Fanuc TP program (LS listing): DISTI_LINE_V10.LS

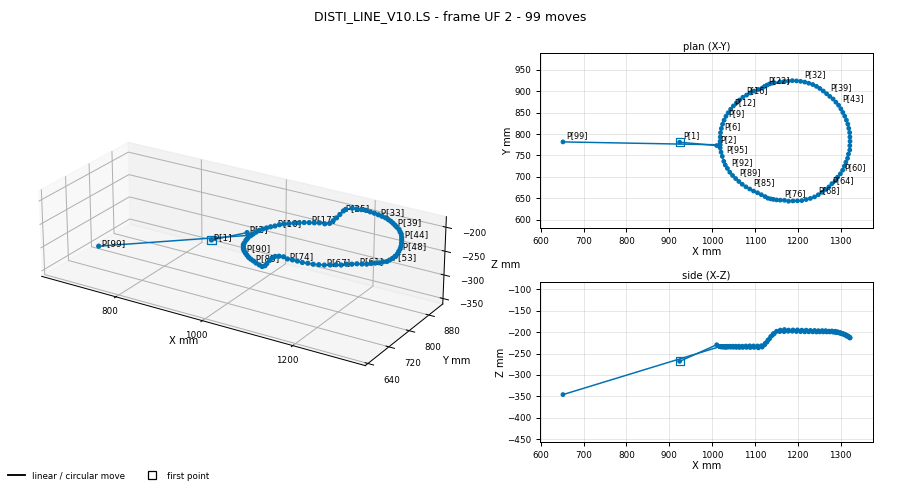
[picture p0: tool path of DISTI_LINE_V10.LS in frame UF 2, 99 of 99 moves have a stored position in this frame; points joined in program order, loops and branches not executed]
/PROG  DISTI_LINE_V10
/ATTR
OWNER		= MNEDITOR;
COMMENT		= "WeldPRO Auto-Gen";
PROG_SIZE	= 7125;
CREATE		= DATE 26-07-31  TIME 11:19:16;
MODIFIED	= DATE 26-07-31  TIME 13:58:52;
FILE_NAME	= DISTI_LI;
VERSION		= 0;
LINE_COUNT	= 113;
MEMORY_SIZE	= 7445;
PROTECT		= READ_WRITE;
TCD:  STACK_SIZE	= 0,
      TASK_PRIORITY	= 50,
      TIME_SLICE	= 0,
      BUSY_LAMP_OFF	= 0,
      ABORT_REQUEST	= 0,
      PAUSE_REQUEST	= 0;
DEFAULT_GROUP	= 1,*,*,*,*;
CONTROL_CODE	= 00000000 00000000;
/APPL
/MN
   1:  !WeldPRO Auto-Generated TPP ;
   2:  !TOR_XL_2026, TOR_xl_2907 ;
   3:   ;
   4:  UFRAME_NUM=2 ;
   5:  UTOOL_NUM=2 ;
   6:  !Feature Approach ;
   7:J P[1] 100% FINE    ;
   8:   ;
   9:  !Segment1 ;
  10:L P[2] 2000mm/sec FINE    ;
  11:   ;
  12:  CALL LASER_OFF    ;
  13:L P[3] R[23:moving]mm/sec CNT100    ;
  14:L P[4] R[23:moving]mm/sec CNT100    ;
  15:L P[5] R[23:moving]mm/sec CNT100    ;
  16:L P[6] R[23:moving]mm/sec CNT100    ;
  17:L P[7] R[23:moving]mm/sec CNT100    ;
  18:L P[8] R[23:moving]mm/sec CNT100    ;
  19:L P[9] R[23:moving]mm/sec CNT100    ;
  20:L P[10] R[23:moving]mm/sec CNT100    ;
  21:L P[11] R[23:moving]mm/sec CNT100    ;
  22:L P[12] R[23:moving]mm/sec CNT100    ;
  23:L P[13] R[23:moving]mm/sec CNT100    ;
  24:L P[14] R[23:moving]mm/sec CNT100    ;
  25:L P[15] R[23:moving]mm/sec CNT100    ;
  26:L P[16] R[23:moving]mm/sec CNT100    ;
  27:L P[17] R[23:moving]mm/sec CNT100    ;
  28:L P[18] R[23:moving]mm/sec CNT100    ;
  29:L P[19] R[23:moving]mm/sec CNT100    ;
  30:L P[20] R[23:moving]mm/sec CNT100    ;
  31:L P[21] R[23:moving]mm/sec CNT100    ;
  32:L P[22] R[23:moving]mm/sec CNT100    ;
  33:L P[23] R[23:moving]mm/sec CNT100    ;
  34:L P[24] R[23:moving]mm/sec CNT100    ;
  35:L P[25] R[23:moving]mm/sec CNT100    ;
  36:L P[26] R[23:moving]mm/sec CNT100    ;
  37:L P[27] R[23:moving]mm/sec CNT100    ;
  38:L P[28] R[23:moving]mm/sec CNT100    ;
  39:L P[29] R[23:moving]mm/sec CNT100    ;
  40:L P[30] R[23:moving]mm/sec CNT100    ;
  41:L P[31] R[23:moving]mm/sec CNT100    ;
  42:L P[32] R[23:moving]mm/sec CNT100    ;
  43:L P[33] R[23:moving]mm/sec CNT100    ;
  44:L P[34] R[23:moving]mm/sec CNT100    ;
  45:L P[35] R[23:moving]mm/sec CNT100    ;
  46:L P[36] R[23:moving]mm/sec CNT100    ;
  47:L P[37] R[23:moving]mm/sec CNT100    ;
  48:L P[38] R[23:moving]mm/sec CNT100    ;
  49:L P[39] R[23:moving]mm/sec CNT100    ;
  50:L P[40] R[23:moving]mm/sec CNT100    ;
  51:L P[41] R[23:moving]mm/sec CNT100    ;
  52:L P[42] R[23:moving]mm/sec CNT100    ;
  53:L P[43] R[23:moving]mm/sec CNT100    ;
  54:L P[44] R[23:moving]mm/sec CNT100    ;
  55:L P[45] R[23:moving]mm/sec CNT100    ;
  56:L P[46] R[23:moving]mm/sec CNT100    ;
  57:L P[47] R[23:moving]mm/sec CNT100    ;
  58:L P[48] R[23:moving]mm/sec CNT100    ;
  59:L P[49] R[23:moving]mm/sec CNT100    ;
  60:L P[50] R[23:moving]mm/sec CNT100    ;
  61:L P[51] R[23:moving]mm/sec CNT100    ;
  62:L P[52] R[23:moving]mm/sec CNT100    ;
  63:L P[53] R[23:moving]mm/sec CNT100    ;
  64:L P[54] R[23:moving]mm/sec CNT100    ;
  65:L P[55] R[23:moving]mm/sec CNT100    ;
  66:L P[56] R[23:moving]mm/sec CNT100    ;
  67:L P[57] R[23:moving]mm/sec CNT100    ;
  68:L P[58] R[23:moving]mm/sec CNT100    ;
  69:L P[59] R[23:moving]mm/sec CNT100    ;
  70:L P[60] R[23:moving]mm/sec CNT100    ;
  71:L P[61] R[23:moving]mm/sec CNT100    ;
  72:L P[62] R[23:moving]mm/sec CNT100    ;
  73:L P[63] R[23:moving]mm/sec CNT100    ;
  74:L P[64] R[23:moving]mm/sec CNT100    ;
  75:L P[65] R[23:moving]mm/sec CNT100    ;
  76:L P[66] R[23:moving]mm/sec CNT100    ;
  77:L P[67] R[23:moving]mm/sec CNT100    ;
  78:L P[68] R[23:moving]mm/sec CNT100    ;
  79:L P[69] R[23:moving]mm/sec CNT100    ;
  80:L P[70] R[23:moving]mm/sec CNT100    ;
  81:L P[71] R[23:moving]mm/sec CNT100    ;
  82:L P[72] R[23:moving]mm/sec CNT100    ;
  83:L P[73] R[23:moving]mm/sec CNT100    ;
  84:L P[74] R[23:moving]mm/sec CNT100    ;
  85:L P[75] R[23:moving]mm/sec CNT100    ;
  86:L P[76] R[23:moving]mm/sec CNT100    ;
  87:L P[77] R[23:moving]mm/sec CNT100    ;
  88:L P[78] R[23:moving]mm/sec CNT100    ;
  89:L P[79] R[23:moving]mm/sec CNT100    ;
  90:L P[80] R[23:moving]mm/sec CNT100    ;
  91:L P[81] R[23:moving]mm/sec CNT100    ;
  92:L P[82] R[23:moving]mm/sec CNT100    ;
  93:L P[83] R[23:moving]mm/sec CNT100    ;
  94:L P[84] R[23:moving]mm/sec CNT100    ;
  95:L P[85] R[23:moving]mm/sec CNT100    ;
  96:L P[86] R[23:moving]mm/sec CNT100    ;
  97:L P[87] R[23:moving]mm/sec CNT100    ;
  98:L P[88] R[23:moving]mm/sec CNT100    ;
  99:L P[89] R[23:moving]mm/sec CNT100    ;
 100:L P[90] R[23:moving]mm/sec CNT100    ;
 101:L P[91] R[23:moving]mm/sec CNT100    ;
 102:L P[92] R[23:moving]mm/sec CNT100    ;
 103:L P[93] R[23:moving]mm/sec CNT100    ;
 104:L P[94] R[23:moving]mm/sec CNT100    ;
 105:L P[95] R[23:moving]mm/sec CNT100    ;
 106:L P[96] R[23:moving]mm/sec CNT100    ;
 107:L P[97] R[23:moving]mm/sec CNT100    ;
 108:L P[98] R[23:moving]mm/sec FINE    ;
 109:  CALL LASER_OFF    ;
 110:   ;
 111:  !Feature Retreat ;
 112:L P[99] 2000mm/sec FINE    ;
 113:  CALL ROTATE    ;
/POS
P[1]{
   GP1:
	UF : 2, UT : 2,		CONFIG : 'F D T, 0, 0, 0',
	X =   924.335  mm,	Y =   780.986  mm,	Z =  -268.284  mm,
	W =  -106.495 deg,	P =   -15.000 deg,	R =    94.234 deg
};
P[2]{
   GP1:
	UF : 2, UT : 2,		CONFIG : 'F D T, 0, 0, 0',
	X =  1011.104  mm,	Y =   773.115  mm,	Z =  -229.520  mm,
	W =  -106.497 deg,	P =   -14.995 deg,	R =    94.216 deg
};
P[3]{
   GP1:
	UF : 2, UT : 2,		CONFIG : 'F D T, 0, 0, 0',
	X =  1018.942  mm,	Y =   775.004  mm,	Z =  -233.963  mm,
	W =  -106.501 deg,	P =   -14.998 deg,	R =    94.232 deg
};
P[4]{
   GP1:
	UF : 2, UT : 2,		CONFIG : 'F D T, 0, 0, 0',
	X =  1018.850  mm,	Y =   783.088  mm,	Z =  -234.009  mm,
	W =  -106.497 deg,	P =   -15.098 deg,	R =    90.375 deg
};
P[5]{
   GP1:
	UF : 2, UT : 2,		CONFIG : 'F D T, 0, 0, 0',
	X =  1019.160  mm,	Y =   793.076  mm,	Z =  -233.945  mm,
	W =  -106.481 deg,	P =   -15.217 deg,	R =    85.597 deg
};
P[6]{
   GP1:
	UF : 2, UT : 2,		CONFIG : 'F D T, 0, 0, 0',
	X =  1019.791  mm,	Y =   803.211  mm,	Z =  -234.335  mm,
	W =  -106.456 deg,	P =   -15.334 deg,	R =    80.807 deg
};
P[7]{
   GP1:
	UF : 2, UT : 2,		CONFIG : 'F D T, 0, 0, 0',
	X =  1021.863  mm,	Y =   813.075  mm,	Z =  -234.445  mm,
	W =  -106.423 deg,	P =   -15.449 deg,	R =    76.083 deg
};
P[8]{
   GP1:
	UF : 2, UT : 2,		CONFIG : 'F D T, 0, 0, 0',
	X =  1024.600  mm,	Y =   822.900  mm,	Z =  -234.958  mm,
	W =  -106.378 deg,	P =   -15.565 deg,	R =    71.217 deg
};
P[9]{
   GP1:
	UF : 2, UT : 2,		CONFIG : 'F D T, 0, 0, 0',
	X =  1028.129  mm,	Y =   832.354  mm,	Z =  -235.228  mm,
	W =  -106.322 deg,	P =   -15.679 deg,	R =    66.207 deg
};
P[10]{
   GP1:
	UF : 2, UT : 2,		CONFIG : 'F D T, 0, 0, 0',
	X =  1032.559  mm,	Y =   841.504  mm,	Z =  -235.811  mm,
	W =  -106.254 deg,	P =   -15.791 deg,	R =    61.015 deg
};
P[11]{
   GP1:
	UF : 2, UT : 2,		CONFIG : 'F D T, 0, 0, 0',
	X =  1037.701  mm,	Y =   849.782  mm,	Z =  -235.048  mm,
	W =  -106.179 deg,	P =   -15.896 deg,	R =    55.983 deg
};
P[12]{
   GP1:
	UF : 2, UT : 2,		CONFIG : 'F D T, 0, 0, 0',
	X =  1043.515  mm,	Y =   857.951  mm,	Z =  -235.221  mm,
	W =  -106.096 deg,	P =   -15.986 deg,	R =    51.162 deg
};
P[13]{
   GP1:
	UF : 2, UT : 2,		CONFIG : 'F D T, 0, 0, 0',
	X =  1049.936  mm,	Y =   865.646  mm,	Z =  -235.476  mm,
	W =  -106.012 deg,	P =   -16.066 deg,	R =    46.632 deg
};
P[14]{
   GP1:
	UF : 2, UT : 2,		CONFIG : 'F D T, 0, 0, 0',
	X =  1056.965  mm,	Y =   872.757  mm,	Z =  -235.696  mm,
	W =  -105.919 deg,	P =   -16.142 deg,	R =    41.952 deg
};
P[15]{
   GP1:
	UF : 2, UT : 2,		CONFIG : 'F D T, 0, 0, 0',
	X =  1064.279  mm,	Y =   879.670  mm,	Z =  -235.896  mm,
	W =  -105.870 deg,	P =   -16.177 deg,	R =    39.609 deg
};
P[16]{
   GP1:
	UF : 2, UT : 2,		CONFIG : 'F D T, 0, 0, 0',
	X =  1071.970  mm,	Y =   885.960  mm,	Z =  -235.776  mm,
	W =  -105.777 deg,	P =   -16.235 deg,	R =    35.365 deg
};
P[17]{
   GP1:
	UF : 2, UT : 2,		CONFIG : 'F D T, 0, 0, 0',
	X =  1080.644  mm,	Y =   890.885  mm,	Z =  -235.790  mm,
	W =  -105.677 deg,	P =   -16.289 deg,	R =    30.964 deg
};
P[18]{
   GP1:
	UF : 2, UT : 2,		CONFIG : 'F D T, 0, 0, 0',
	X =  1089.333  mm,	Y =   895.820  mm,	Z =  -236.037  mm,
	W =  -105.579 deg,	P =   -16.333 deg,	R =    26.830 deg
};
P[19]{
   GP1:
	UF : 2, UT : 2,		CONFIG : 'F D T, 0, 0, 0',
	X =  1098.139  mm,	Y =   900.305  mm,	Z =  -235.787  mm,
	W =  -105.536 deg,	P =   -16.344 deg,	R =    25.018 deg
};
P[20]{
   GP1:
	UF : 2, UT : 2,		CONFIG : 'F D T, 0, 0, 0',
	X =  1108.071  mm,	Y =   904.161  mm,	Z =  -236.936  mm,
	W =  -116.027 deg,	P =   -16.063 deg,	R =    30.267 deg
};
P[21]{
   GP1:
	UF : 2, UT : 2,		CONFIG : 'F D T, 0, 0, 0',
	X =  1117.118  mm,	Y =   907.345  mm,	Z =  -235.084  mm,
	W =  -126.877 deg,	P =   -15.356 deg,	R =    25.893 deg
};
P[22]{
   GP1:
	UF : 2, UT : 2,		CONFIG : 'F D T, 0, 0, 0',
	X =  1122.637  mm,	Y =   911.322  mm,	Z =  -229.837  mm,
	W =  -119.393 deg,	P =   -15.981 deg,	R =    16.221 deg
};
P[23]{
   GP1:
	UF : 2, UT : 2,		CONFIG : 'F D T, 0, 0, 0',
	X =  1128.381  mm,	Y =   914.380  mm,	Z =  -223.360  mm,
	W =  -115.329 deg,	P =   -16.208 deg,	R =    11.788 deg
};
P[24]{
   GP1:
	UF : 2, UT : 2,		CONFIG : 'F D T, 0, 0, 0',
	X =  1134.187  mm,	Y =   916.917  mm,	Z =  -215.853  mm,
	W =  -112.639 deg,	P =   -16.315 deg,	R =     9.714 deg
};
P[25]{
   GP1:
	UF : 2, UT : 2,		CONFIG : 'F D T, 0, 0, 0',
	X =  1140.842  mm,	Y =   918.847  mm,	Z =  -207.606  mm,
	W =  -110.015 deg,	P =   -16.386 deg,	R =     9.649 deg
};
P[26]{
   GP1:
	UF : 2, UT : 2,		CONFIG : 'F D T, 0, 0, 0',
	X =  1145.182  mm,	Y =   919.975  mm,	Z =  -203.759  mm,
	W =  -108.552 deg,	P =   -16.418 deg,	R =     8.950 deg
};
P[27]{
   GP1:
	UF : 2, UT : 2,		CONFIG : 'F D T, 0, 0, 0',
	X =  1158.300  mm,	Y =   922.045  mm,	Z =  -198.881  mm,
	W =  -105.409 deg,	P =   -16.443 deg,	R =     6.805 deg
};
P[28]{
   GP1:
	UF : 2, UT : 2,		CONFIG : 'F D T, 0, 0, 0',
	X =  1168.271  mm,	Y =   922.879  mm,	Z =  -198.949  mm,
	W =  -104.866 deg,	P =   -16.444 deg,	R =     5.597 deg
};
P[29]{
   GP1:
	UF : 2, UT : 2,		CONFIG : 'F D T, 0, 0, 0',
	X =  1177.818  mm,	Y =   923.489  mm,	Z =  -198.132  mm,
	W =  -104.887 deg,	P =   -16.444 deg,	R =     3.523 deg
};
P[30]{
   GP1:
	UF : 2, UT : 2,		CONFIG : 'F D T, 0, 0, 0',
	X =  1187.403  mm,	Y =   924.750  mm,	Z =  -198.093  mm,
	W =  -104.930 deg,	P =   -16.439 deg,	R =     -.729 deg
};
P[31]{
   GP1:
	UF : 2, UT : 2,		CONFIG : 'F D T, 0, 0, 0',
	X =  1197.178  mm,	Y =   924.128  mm,	Z =  -198.675  mm,
	W =  -104.979 deg,	P =   -16.424 deg,	R =    -5.541 deg
};
P[32]{
   GP1:
	UF : 2, UT : 2,		CONFIG : 'F D T, 0, 0, 0',
	X =  1206.835  mm,	Y =   923.072  mm,	Z =  -198.951  mm,
	W =  -105.028 deg,	P =   -16.400 deg,	R =   -10.259 deg
};
P[33]{
   GP1:
	UF : 2, UT : 2,		CONFIG : 'F D T, 0, 0, 0',
	X =  1216.484  mm,	Y =   921.355  mm,	Z =  -199.461  mm,
	W =  -105.070 deg,	P =   -16.371 deg,	R =   -14.490 deg
};
P[34]{
   GP1:
	UF : 2, UT : 2,		CONFIG : 'F D T, 0, 0, 0',
	X =  1225.848  mm,	Y =   918.697  mm,	Z =  -199.382  mm,
	W =  -105.112 deg,	P =   -16.334 deg,	R =   -18.515 deg
};
P[35]{
   GP1:
	UF : 2, UT : 2,		CONFIG : 'F D T, 0, 0, 0',
	X =  1235.082  mm,	Y =   915.694  mm,	Z =  -199.428  mm,
	W =  -105.158 deg,	P =   -16.285 deg,	R =   -23.051 deg
};
P[36]{
   GP1:
	UF : 2, UT : 2,		CONFIG : 'F D T, 0, 0, 0',
	X =  1243.756  mm,	Y =   911.418  mm,	Z =  -199.733  mm,
	W =  -105.219 deg,	P =   -16.204 deg,	R =   -29.417 deg
};
P[37]{
   GP1:
	UF : 2, UT : 2,		CONFIG : 'F D T, 0, 0, 0',
	X =  1251.633  mm,	Y =   906.491  mm,	Z =  -199.508  mm,
	W =  -105.311 deg,	P =   -16.047 deg,	R =   -39.415 deg
};
P[38]{
   GP1:
	UF : 2, UT : 2,		CONFIG : 'F D T, 0, 0, 0',
	X =  1259.725  mm,	Y =   900.526  mm,	Z =  -199.596  mm,
	W =  -105.307 deg,	P =   -16.055 deg,	R =   -38.974 deg
};
P[39]{
   GP1:
	UF : 2, UT : 2,		CONFIG : 'F D T, 0, 0, 0',
	X =  1267.493  mm,	Y =   894.217  mm,	Z =  -199.670  mm,
	W =  -105.302 deg,	P =   -16.063 deg,	R =   -38.625 deg
};
P[40]{
   GP1:
	UF : 2, UT : 2,		CONFIG : 'F D T, 0, 0, 0',
	X =  1274.833  mm,	Y =   887.985  mm,	Z =  -199.664  mm,
	W =  -105.469 deg,	P =   -15.944 deg,	R =   -44.976 deg
};
P[41]{
   GP1:
	UF : 2, UT : 2,		CONFIG : 'F D T, 0, 0, 0',
	X =  1282.713  mm,	Y =   881.925  mm,	Z =  -200.195  mm,
	W =  -105.661 deg,	P =   -15.890 deg,	R =   -47.714 deg
};
P[42]{
   GP1:
	UF : 2, UT : 2,		CONFIG : 'F D T, 0, 0, 0',
	X =  1289.091  mm,	Y =   874.515  mm,	Z =  -201.203  mm,
	W =  -106.210 deg,	P =   -15.792 deg,	R =   -52.259 deg
};
P[43]{
   GP1:
	UF : 2, UT : 2,		CONFIG : 'F D T, 0, 0, 0',
	X =  1295.469  mm,	Y =   867.345  mm,	Z =  -201.768  mm,
	W =  -106.927 deg,	P =   -15.688 deg,	R =   -56.663 deg
};
P[44]{
   GP1:
	UF : 2, UT : 2,		CONFIG : 'F D T, 0, 0, 0',
	X =  1300.802  mm,	Y =   858.976  mm,	Z =  -203.772  mm,
	W =  -107.603 deg,	P =   -15.597 deg,	R =   -60.243 deg
};
P[45]{
   GP1:
	UF : 2, UT : 2,		CONFIG : 'F D T, 0, 0, 0',
	X =  1305.393  mm,	Y =   850.522  mm,	Z =  -204.867  mm,
	W =  -108.271 deg,	P =   -15.504 deg,	R =   -63.686 deg
};
P[46]{
   GP1:
	UF : 2, UT : 2,		CONFIG : 'F D T, 0, 0, 0',
	X =  1309.903  mm,	Y =   841.761  mm,	Z =  -206.715  mm,
	W =  -109.143 deg,	P =   -15.377 deg,	R =   -68.203 deg
};
P[47]{
   GP1:
	UF : 2, UT : 2,		CONFIG : 'F D T, 0, 0, 0',
	X =  1313.877  mm,	Y =   832.536  mm,	Z =  -208.918  mm,
	W =  -109.899 deg,	P =   -15.253 deg,	R =   -72.505 deg
};
P[48]{
   GP1:
	UF : 2, UT : 2,		CONFIG : 'F D T, 0, 0, 0',
	X =  1317.069  mm,	Y =   823.150  mm,	Z =  -210.301  mm,
	W =  -110.273 deg,	P =   -15.181 deg,	R =   -74.981 deg
};
P[49]{
   GP1:
	UF : 2, UT : 2,		CONFIG : 'F D T, 0, 0, 0',
	X =  1319.251  mm,	Y =   813.364  mm,	Z =  -211.544  mm,
	W =  -110.635 deg,	P =   -14.305 deg,	R =   -78.232 deg
};
P[50]{
   GP1:
	UF : 2, UT : 2,		CONFIG : 'F D T, 0, 0, 0',
	X =  1321.365  mm,	Y =   803.425  mm,	Z =  -212.773  mm,
	W =  -111.054 deg,	P =   -14.769 deg,	R =   -83.164 deg
};
P[51]{
   GP1:
	UF : 2, UT : 2,		CONFIG : 'F D T, 0, 0, 0',
	X =  1321.943  mm,	Y =   793.209  mm,	Z =  -213.629  mm,
	W =  -111.190 deg,	P =   -15.305 deg,	R =   -88.308 deg
};
P[52]{
   GP1:
	UF : 2, UT : 2,		CONFIG : 'F D T, 0, 0, 0',
	X =  1322.253  mm,	Y =   783.157  mm,	Z =  -213.410  mm,
	W =  -111.129 deg,	P =   -15.645 deg,	R =   -91.614 deg
};
P[53]{
   GP1:
	UF : 2, UT : 2,		CONFIG : 'F D T, 0, 0, 0',
	X =  1321.706  mm,	Y =   772.971  mm,	Z =  -213.015  mm,
	W =  -110.757 deg,	P =   -14.624 deg,	R =   -96.575 deg
};
P[54]{
   GP1:
	UF : 2, UT : 2,		CONFIG : 'F D T, 0, 0, 0',
	X =  1321.590  mm,	Y =   762.769  mm,	Z =  -212.022  mm,
	W =  -110.276 deg,	P =   -14.535 deg,	R =  -100.836 deg
};
P[55]{
   GP1:
	UF : 2, UT : 2,		CONFIG : 'F D T, 0, 0, 0',
	X =  1318.584  mm,	Y =   753.304  mm,	Z =  -209.863  mm,
	W =  -109.635 deg,	P =   -14.447 deg,	R =  -105.265 deg
};
P[56]{
   GP1:
	UF : 2, UT : 2,		CONFIG : 'F D T, 0, 0, 0',
	X =  1316.464  mm,	Y =   743.431  mm,	Z =  -208.514  mm,
	W =  -109.083 deg,	P =   -14.382 deg,	R =  -108.626 deg
};
P[57]{
   GP1:
	UF : 2, UT : 2,		CONFIG : 'F D T, 0, 0, 0',
	X =  1312.561  mm,	Y =   734.284  mm,	Z =  -206.441  mm,
	W =  -108.349 deg,	P =   -14.302 deg,	R =  -112.873 deg
};
P[58]{
   GP1:
	UF : 2, UT : 2,		CONFIG : 'F D T, 0, 0, 0',
	X =  1308.951  mm,	Y =   724.963  mm,	Z =  -204.585  mm,
	W =  -107.748 deg,	P =   -14.239 deg,	R =  -116.265 deg
};
P[59]{
   GP1:
	UF : 2, UT : 2,		CONFIG : 'F D T, 0, 0, 0',
	X =  1304.942  mm,	Y =   715.581  mm,	Z =  -203.183  mm,
	W =  -106.924 deg,	P =   -14.148 deg,	R =  -121.191 deg
};
P[60]{
   GP1:
	UF : 2, UT : 2,		CONFIG : 'F D T, 0, 0, 0',
	X =  1299.663  mm,	Y =   707.136  mm,	Z =  -201.022  mm,
	W =  -106.269 deg,	P =   -14.066 deg,	R =  -125.698 deg
};
P[61]{
   GP1:
	UF : 2, UT : 2,		CONFIG : 'F D T, 0, 0, 0',
	X =  1293.247  mm,	Y =   699.470  mm,	Z =  -199.153  mm,
	W =  -105.781 deg,	P =   -13.988 deg,	R =  -130.143 deg
};
P[62]{
   GP1:
	UF : 2, UT : 2,		CONFIG : 'F D T, 0, 0, 0',
	X =  1287.561  mm,	Y =   690.909  mm,	Z =  -197.986  mm,
	W =  -105.526 deg,	P =   -13.913 deg,	R =  -134.519 deg
};
P[63]{
   GP1:
	UF : 2, UT : 2,		CONFIG : 'F D T, 0, 0, 0',
	X =  1279.931  mm,	Y =   684.263  mm,	Z =  -197.327  mm,
	W =  -105.437 deg,	P =   -13.849 deg,	R =  -138.629 deg
};
P[64]{
   GP1:
	UF : 2, UT : 2,		CONFIG : 'F D T, 0, 0, 0',
	X =  1272.996  mm,	Y =   676.712  mm,	Z =  -197.730  mm,
	W =  -105.429 deg,	P =   -13.831 deg,	R =  -139.837 deg
};
P[65]{
   GP1:
	UF : 2, UT : 2,		CONFIG : 'F D T, 0, 0, 0',
	X =  1265.430  mm,	Y =   670.792  mm,	Z =  -196.653  mm,
	W =  -105.443 deg,	P =   -13.863 deg,	R =  -137.727 deg
};
P[66]{
   GP1:
	UF : 2, UT : 2,		CONFIG : 'F D T, 0, 0, 0',
	X =  1257.252  mm,	Y =   663.987  mm,	Z =  -196.494  mm,
	W =  -105.373 deg,	P =   -13.729 deg,	R =  -147.436 deg
};
P[67]{
   GP1:
	UF : 2, UT : 2,		CONFIG : 'F D T, 0, 0, 0',
	X =  1248.165  mm,	Y =   658.329  mm,	Z =  -196.704  mm,
	W =  -105.298 deg,	P =   -13.637 deg,	R =  -156.529 deg
};
P[68]{
   GP1:
	UF : 2, UT : 2,		CONFIG : 'F D T, 0, 0, 0',
	X =  1239.358  mm,	Y =   653.310  mm,	Z =  -196.157  mm,
	W =  -105.277 deg,	P =   -13.618 deg,	R =  -158.976 deg
};
P[69]{
   GP1:
	UF : 2, UT : 2,		CONFIG : 'F D T, 0, 0, 0',
	X =  1229.649  mm,	Y =   649.730  mm,	Z =  -196.118  mm,
	W =  -105.241 deg,	P =   -13.592 deg,	R =  -162.969 deg
};
P[70]{
   GP1:
	UF : 2, UT : 2,		CONFIG : 'F D T, 0, 0, 0',
	X =  1219.769  mm,	Y =   647.170  mm,	Z =  -195.496  mm,
	W =  -105.203 deg,	P =   -13.573 deg,	R =  -167.022 deg
};
P[71]{
   GP1:
	UF : 2, UT : 2,		CONFIG : 'F D T, 0, 0, 0',
	X =  1209.672  mm,	Y =   644.649  mm,	Z =  -195.520  mm,
	W =  -105.159 deg,	P =   -13.560 deg,	R =  -171.569 deg
};
P[72]{
   GP1:
	UF : 2, UT : 2,		CONFIG : 'F D T, 0, 0, 0',
	X =  1199.433  mm,	Y =   644.195  mm,	Z =  -194.880  mm,
	W =  -105.113 deg,	P =   -13.556 deg,	R =  -176.312 deg
};
P[73]{
   GP1:
	UF : 2, UT : 2,		CONFIG : 'F D T, 0, 0, 0',
	X =  1189.086  mm,	Y =   643.937  mm,	Z =  -195.031  mm,
	W =  -105.068 deg,	P =   -13.561 deg,	R =   179.213 deg
};
P[74]{
   GP1:
	UF : 2, UT : 2,		CONFIG : 'F D T, 0, 0, 0',
	X =  1178.770  mm,	Y =   643.156  mm,	Z =  -195.259  mm,
	W =  -105.038 deg,	P =   -13.569 deg,	R =   176.231 deg
};
P[75]{
   GP1:
	UF : 2, UT : 2,		CONFIG : 'F D T, 0, 0, 0',
	X =  1169.122  mm,	Y =   645.376  mm,	Z =  -194.039  mm,
	W =  -105.207 deg,	P =   -13.572 deg,	R =   175.290 deg
};
P[76]{
   GP1:
	UF : 2, UT : 2,		CONFIG : 'F D T, 0, 0, 0',
	X =  1159.384  mm,	Y =   645.670  mm,	Z =  -195.292  mm,
	W =  -107.012 deg,	P =   -13.569 deg,	R =   174.537 deg
};
P[77]{
   GP1:
	UF : 2, UT : 2,		CONFIG : 'F D T, 0, 0, 0',
	X =  1150.691  mm,	Y =   646.290  mm,	Z =  -198.036  mm,
	W =  -109.414 deg,	P =   -13.538 deg,	R =   174.483 deg
};
P[78]{
   GP1:
	UF : 2, UT : 2,		CONFIG : 'F D T, 0, 0, 0',
	X =  1143.181  mm,	Y =   647.458  mm,	Z =  -203.547  mm,
	W =  -112.196 deg,	P =   -13.466 deg,	R =   175.323 deg
};
P[79]{
   GP1:
	UF : 2, UT : 2,		CONFIG : 'F D T, 0, 0, 0',
	X =  1137.079  mm,	Y =   648.698  mm,	Z =  -210.369  mm,
	W =  -114.872 deg,	P =   -13.369 deg,	R =   175.422 deg
};
P[80]{
   GP1:
	UF : 2, UT : 2,		CONFIG : 'F D T, 0, 0, 0',
	X =  1130.436  mm,	Y =   650.205  mm,	Z =  -218.773  mm,
	W =  -120.114 deg,	P =   -13.109 deg,	R =   172.293 deg
};
P[81]{
   GP1:
	UF : 2, UT : 2,		CONFIG : 'F D T, 0, 0, 0',
	X =  1123.985  mm,	Y =   654.011  mm,	Z =  -226.383  mm,
	W =  -126.809 deg,	P =   -12.620 deg,	R =   167.791 deg
};
P[82]{
   GP1:
	UF : 2, UT : 2,		CONFIG : 'F D T, 0, 0, 0',
	X =  1115.177  mm,	Y =   658.431  mm,	Z =  -231.762  mm,
	W =  -119.561 deg,	P =   -13.285 deg,	R =   157.806 deg
};
P[83]{
   GP1:
	UF : 2, UT : 2,		CONFIG : 'F D T, 0, 0, 0',
	X =  1106.207  mm,	Y =   663.031  mm,	Z =  -232.341  mm,
	W =  -107.325 deg,	P =   -13.741 deg,	R =   154.437 deg
};
P[84]{
   GP1:
	UF : 2, UT : 2,		CONFIG : 'F D T, 0, 0, 0',
	X =  1096.909  mm,	Y =   666.875  mm,	Z =  -232.283  mm,
	W =  -105.746 deg,	P =   -13.749 deg,	R =   154.142 deg
};
P[85]{
   GP1:
	UF : 2, UT : 2,		CONFIG : 'F D T, 0, 0, 0',
	X =  1088.043  mm,	Y =   671.716  mm,	Z =  -232.065  mm,
	W =  -105.804 deg,	P =   -13.784 deg,	R =   151.506 deg
};
P[86]{
   GP1:
	UF : 2, UT : 2,		CONFIG : 'F D T, 0, 0, 0',
	X =  1079.090  mm,	Y =   676.830  mm,	Z =  -232.437  mm,
	W =  -105.885 deg,	P =   -13.838 deg,	R =   147.739 deg
};
P[87]{
   GP1:
	UF : 2, UT : 2,		CONFIG : 'F D T, 0, 0, 0',
	X =  1070.535  mm,	Y =   682.786  mm,	Z =  -232.933  mm,
	W =  -105.988 deg,	P =   -13.918 deg,	R =   142.681 deg
};
P[88]{
   GP1:
	UF : 2, UT : 2,		CONFIG : 'F D T, 0, 0, 0',
	X =  1062.634  mm,	Y =   689.354  mm,	Z =  -232.781  mm,
	W =  -106.084 deg,	P =   -14.001 deg,	R =   137.677 deg
};
P[89]{
   GP1:
	UF : 2, UT : 2,		CONFIG : 'F D T, 0, 0, 0',
	X =  1055.198  mm,	Y =   696.163  mm,	Z =  -232.905  mm,
	W =  -106.129 deg,	P =   -14.056 deg,	R =   135.014 deg
};
P[90]{
   GP1:
	UF : 2, UT : 2,		CONFIG : 'F D T, 0, 0, 0',
	X =  1047.955  mm,	Y =   703.329  mm,	Z =  -232.932  mm,
	W =  -106.186 deg,	P =   -14.117 deg,	R =   131.622 deg
};
P[91]{
   GP1:
	UF : 2, UT : 2,		CONFIG : 'F D T, 0, 0, 0',
	X =  1041.505  mm,	Y =   710.845  mm,	Z =  -233.012  mm,
	W =  -106.269 deg,	P =   -14.234 deg,	R =   126.207 deg
};
P[92]{
   GP1:
	UF : 2, UT : 2,		CONFIG : 'F D T, 0, 0, 0',
	X =  1035.939  mm,	Y =   719.763  mm,	Z =  -233.106  mm,
	W =  -106.343 deg,	P =   -14.367 deg,	R =   120.225 deg
};
P[93]{
   GP1:
	UF : 2, UT : 2,		CONFIG : 'F D T, 0, 0, 0',
	X =  1030.975  mm,	Y =   727.661  mm,	Z =  -233.336  mm,
	W =  -106.383 deg,	P =   -14.448 deg,	R =   116.672 deg
};
P[94]{
   GP1:
	UF : 2, UT : 2,		CONFIG : 'F D T, 0, 0, 0',
	X =  1027.536  mm,	Y =   736.304  mm,	Z =  -233.837  mm,
	W =  -106.433 deg,	P =   -14.556 deg,	R =   111.957 deg
};
P[95]{
   GP1:
	UF : 2, UT : 2,		CONFIG : 'F D T, 0, 0, 0',
	X =  1023.984  mm,	Y =   747.963  mm,	Z =  -233.467  mm,
	W =  -106.465 deg,	P =   -14.714 deg,	R =   105.666 deg
};
P[96]{
   GP1:
	UF : 2, UT : 2,		CONFIG : 'F D T, 0, 1, 0',
	X =  1021.138  mm,	Y =   757.780  mm,	Z =  -234.038  mm,
	W =  -106.480 deg,	P =   -14.798 deg,	R =   102.261 deg
};
P[97]{
   GP1:
	UF : 2, UT : 2,		CONFIG : 'F D T, 0, 1, 0',
	X =  1019.006  mm,	Y =   767.672  mm,	Z =  -233.868  mm,
	W =  -106.494 deg,	P =   -14.935 deg,	R =    96.827 deg
};
P[98]{
   GP1:
	UF : 2, UT : 2,		CONFIG : 'F D T, 0, 1, 0',
	X =  1018.391  mm,	Y =   774.925  mm,	Z =  -233.928  mm,
	W =  -106.501 deg,	P =   -15.000 deg,	R =    94.235 deg
};
P[99]{
   GP1:
	UF : 2, UT : 2,		CONFIG : 'F D T, 0, 1, 0',
	X =   651.995  mm,	Y =   781.694  mm,	Z =  -345.952  mm,
	W =  -106.495 deg,	P =   -15.000 deg,	R =    94.234 deg
};
/END
